Yaskawa INFORM job: aruba_21-06-23_cylinder_program.JBI

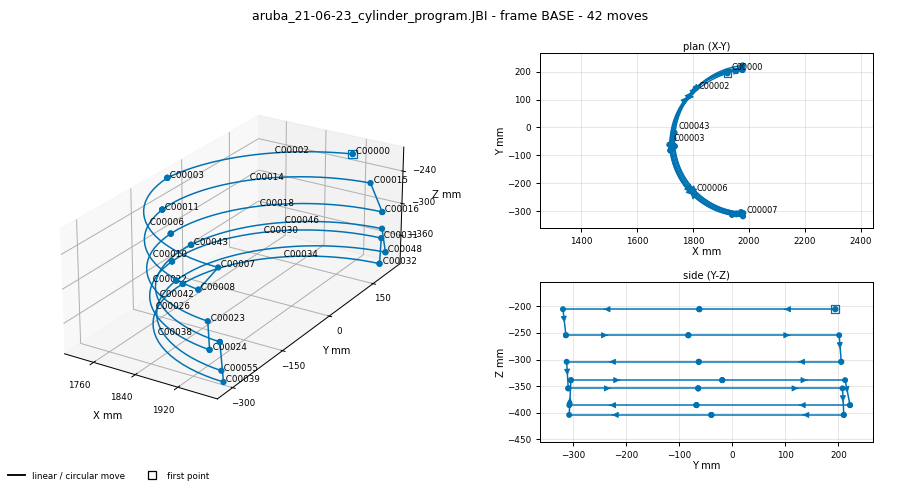
[picture p0: tool path of aruba_21-06-23_cylinder_program.JBI in frame BASE, 42 of 66 moves have a stored position in this frame; points joined in program order, loops and branches not executed]
/JOB
//NAME aruba_21-06-23_cylinder_program
//POS
///NPOS 56,0,56,0,0,0
///TOOL 0
///POSTYPE BASE
///RECTAN
///RCONF 0,0,0,0,0,0,0,0,0,0,0,0,0,0,0,0,0,0,0,0,0,0,0,0
C00000=1923.045603,194.185144,-205.339000,104.153586,-90.000000,5.000000
C00001=1923.045603,194.185144,-205.339000,104.153586,-90.000000,5.000000
C00002=1804.976796,125.705268,-205.339000,135.759368,-90.000000,5.000000
C00003=1715.647484,-61.822449,-205.339000,-177.267001,-90.000000,5.000000
C00004=1715.647484,-61.822449,-205.339000,-177.267001,-90.000000,5.000000
C00005=1715.647484,-61.822449,-205.339000,-177.267001,-90.000000,5.000000
C00006=1797.702002,-242.116782,-205.339000,-134.026420,-90.000000,5.000000
C00007=1978.828028,-318.490725,-205.339000,-91.178076,-90.000000,5.000000
C00008=1939.355207,-312.931172,-254.305000,-99.678760,-90.000000,5.000000
C00009=1939.355207,-312.931172,-254.305000,-99.678760,-90.000000,5.000000
C00010=1808.920889,-251.834088,-254.305000,-130.858681,-90.000000,5.000000
C00011=1718.475494,-82.460121,-254.305000,-172.826486,-90.000000,5.000000
C00012=1718.475494,-82.460121,-254.305000,-172.826486,-90.000000,5.000000
C00013=1718.475494,-82.460121,-254.305000,-172.826486,-90.000000,5.000000
C00014=1770.440864,99.914246,-254.305000,145.159509,-90.000000,5.000000
C00015=1954.941306,201.470356,-254.305000,96.701312,-90.000000,5.000000
C00016=1976.986392,205.347038,-304.305000,91.662845,-90.000000,5.000000
C00017=1976.986392,205.347038,-304.305000,91.662845,-90.000000,5.000000
C00018=1782.331849,112.836364,-304.305000,141.305531,-90.000000,5.000000
C00019=1721.577337,-62.848503,-304.305000,-176.982297,-90.000000,5.000000
C00020=1721.577337,-62.848503,-304.305000,-176.982297,-90.000000,5.000000
C00021=1721.577337,-62.848503,-304.305000,-176.982297,-90.000000,5.000000
C00022=1799.875039,-240.142404,-304.305000,-133.985381,-90.000000,5.000000
C00023=1955.017310,-311.527546,-304.305000,-96.379505,-90.000000,5.000000
C00024=1956.119430,-308.550767,-354.305000,-96.211728,-90.000000,5.000000
C00025=1956.119430,-308.550767,-354.305000,-96.211728,-90.000000,5.000000
C00026=1799.399404,-233.758072,-354.305000,-135.032113,-90.000000,5.000000
C00027=1723.947790,-63.923001,-354.305000,-176.719198,-89.999999,5.000000
C00028=1723.947790,-63.923001,-354.305000,-176.719198,-89.999999,5.000000
C00029=1723.947790,-63.923001,-354.305000,-176.719198,-89.999999,5.000000
C00030=1787.809841,118.598419,-354.305000,139.548090,-90.000000,5.000000
C00031=1975.293908,207.736337,-354.305000,92.024708,-90.000000,5.000000
C00032=1972.059515,210.141000,-404.305000,92.719845,-90.000000,5.000000
C00033=1972.059515,210.141000,-404.305000,92.719845,-90.000000,5.000000
C00034=1813.218693,143.735953,-404.305000,131.606155,-90.000000,5.000000
C00035=1728.847771,-39.166710,-404.305000,177.797354,-90.000000,5.000000
C00036=1728.847771,-39.166710,-404.305000,177.797354,-90.000000,5.000000
C00037=1728.847771,-39.166710,-404.305000,177.797354,-90.000000,5.000000
C00038=1797.953197,-225.866944,-404.305000,-136.504965,-90.000000,5.000000
C00039=1980.178864,-306.786574,-404.305000,-90.931423,-89.999999,5.000000
C00040=1971.675106,-303.470598,-338.834946,180.000000,-60.000000,87.144086
C00041=1971.675106,-303.470598,-338.834946,180.000000,-60.000000,87.144086
C00042=1799.252371,-219.804430,-338.834946,180.000000,-60.000000,42.698011
C00043=1732.800272,-18.639284,-338.834946,180.000000,-60.000000,-6.880276
C00044=1732.800272,-18.639284,-338.834946,180.000000,-60.000000,-6.880276
C00045=1732.800272,-18.639284,-338.834946,180.000000,-60.000000,-6.880276
C00046=1813.665905,143.976915,-338.834946,180.000000,-60.000000,-48.503792
C00047=1973.577851,212.659895,-338.834946,180.000000,-60.000000,-87.638129
C00048=1976.736655,221.903548,-385.887946,-180.000000,-60.000000,-88.385952
C00049=1976.736655,221.903548,-385.887946,-180.000000,-60.000000,-88.385952
C00050=1802.145499,131.858434,-385.887946,180.000000,-60.000000,-44.783591
C00051=1733.939450,-67.253131,-385.887946,180.000000,-60.000000,4.169952
C00052=1733.939450,-67.253131,-385.887946,180.000000,-60.000000,4.169952
C00053=1733.939450,-67.253131,-385.887946,180.000000,-60.000000,4.169952
C00054=1813.069204,-232.815403,-385.887946,180.000000,-60.000000,47.019142
C00055=1976.278956,-306.501347,-385.887946,-180.000000,-60.000000,88.200317
///POSTYPE PULSE
///PULSE
EX00000=92160
EX00001=184320
EX00002=276480
EX00003=368640
///POSTYPE PULSE
///PULSE
EC00000=0
EC00001=0
EC00002=0
EC00003=0
EC00004=0
EC00005=0
EC00006=0
EC00007=0
EC00008=0
EC00009=0
EC00010=0
EC00011=0
EC00012=0
EC00013=0
EC00014=0
EC00015=0
EC00016=0
EC00017=0
EC00018=0
EC00019=0
EC00020=0
EC00021=0
EC00022=0
EC00023=0
EC00024=0
EC00025=0
EC00026=0
EC00027=0
EC00028=0
EC00029=0
EC00030=0
EC00031=0
EC00032=0
EC00033=0
EC00034=0
EC00035=0
EC00036=0
EC00037=0
EC00038=0
EC00039=0
EC00040=0
EC00041=0
EC00042=0
EC00043=0
EC00044=0
EC00045=0
EC00046=0
EC00047=0
EC00048=0
EC00049=0
EC00050=0
EC00051=0
EC00052=0
EC00053=0
EC00054=0
EC00055=0
//INST
///DATE 2023/06/26 11:09
///ATTR SC,RW,RJ
////FRAME BASE
///GROUP1 RB1,ST1
NOP
MOVJ P009 EX000 VJ=15.00
MOVJ P009 VJ=15.00
MOVJ C00000 EC00000 VJ=15.0
CALL JOB:SPYON
MOVC C00001 EC00001 V=150.0
MOVC C00002 EC00002 V=150.0
MOVC C00003 EC00003 V=150.0
MOVL C00004 EC00004 V=150.0
MOVC C00005 EC00005 V=150.0
MOVC C00006 EC00006 V=150.0
MOVC C00007 EC00007 V=150.0
MOVL C00008 EC00008 V=150.0
MOVC C00009 EC00009 V=150.0
MOVC C00010 EC00010 V=150.0
MOVC C00011 EC00011 V=150.0
MOVL C00012 EC00012 V=150.0
MOVC C00013 EC00013 V=150.0
MOVC C00014 EC00014 V=150.0
MOVC C00015 EC00015 V=150.0
MOVL C00016 EC00016 V=150.0
MOVC C00017 EC00017 V=150.0
MOVC C00018 EC00018 V=150.0
MOVC C00019 EC00019 V=150.0
MOVL C00020 EC00020 V=150.0
MOVC C00021 EC00021 V=150.0
MOVC C00022 EC00022 V=150.0
MOVC C00023 EC00023 V=150.0
MOVL C00024 EC00024 V=150.0
MOVC C00025 EC00025 V=150.0
MOVC C00026 EC00026 V=150.0
MOVC C00027 EC00027 V=150.0
MOVL C00028 EC00028 V=150.0
MOVC C00029 EC00029 V=150.0
MOVC C00030 EC00030 V=150.0
MOVC C00031 EC00031 V=150.0
MOVL C00032 EC00032 V=150.0
MOVC C00033 EC00033 V=150.0
MOVC C00034 EC00034 V=150.0
MOVC C00035 EC00035 V=150.0
MOVL C00036 EC00036 V=150.0
MOVC C00037 EC00037 V=150.0
MOVC C00038 EC00038 V=150.0
MOVC C00039 EC00039 V=150.0
MOVL C00040 EC00040 V=150.0
MOVC C00041 EC00041 V=150.0
MOVC C00042 EC00042 V=150.0
MOVC C00043 EC00043 V=150.0
MOVL C00044 EC00044 V=150.0
MOVC C00045 EC00045 V=150.0
MOVC C00046 EC00046 V=150.0
MOVC C00047 EC00047 V=150.0
MOVL C00048 EC00048 V=150.0
MOVC C00049 EC00049 V=150.0
MOVC C00050 EC00050 V=150.0
MOVC C00051 EC00051 V=150.0
MOVL C00052 EC00052 V=150.0
MOVC C00053 EC00053 V=150.0
MOVC C00054 EC00054 V=150.0
MOVC C00055 EC00055 V=150.0
CALL JOB:SPYOF
MOVJ P009 VJ=15.00
MOVL P009 EX00000 V=150.0
MOVJ P009 VJ=15.00
MOVL P009 EX00001 V=150.0
MOVJ P009 VJ=15.00
MOVL P009 EX00002 V=150.0
MOVJ P009 VJ=15.00
MOVL P009 EX00003 V=150.0
END
